{attribute 'GeneratedUsingTerminal: EL3773-0000-0019'}
{attribute addProperty BoxType "EL3773-0000-0019"}
{attribute addProperty Id "U3_SamplesAT %I*U3_Samples_2549228720"}
{attribute addProperty CRC "1711951775"}
{attribute addProperty Size "20"}
TYPE L3_Voltage_Samples_660A4F9F :
STRUCT
	{attribute addProperty Name "U3_Samples"}
	U3_Samples AT %I* : U3_Samples_25492287;
END_STRUCT
END_TYPE

(* stored: Version 1.2.0.0, ProductVersion 3.1.4024.9
   DUT L3_Voltage_Samples_660A4F9F: Id {89204f0e-3290-4eea-b0d3-b7df85452e2c} *)
